Universal Robots PolyScope program: cov st move test.urp

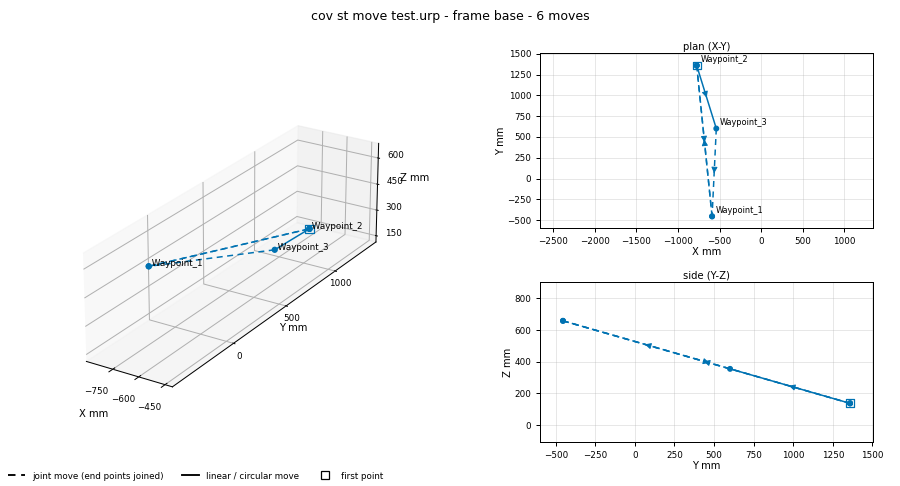
[picture p0: tool path of cov st move test.urp in frame base, 6 of 6 moves have a stored position in this frame; points joined in program order, loops and branches not executed]
Program cov st move test (installation=default directory=/programs createdIn=5.21.3 lastSavedIn=5.21.3 robotSerialNumber=20246801938)
Calibrated DH parameters: a=[-0.000071, -0.790281, -0.600694, 0.000061, -0.000039, 0]; d=[0.236272, 604.465945, 132.116513, -736.382239, 0.159268, 0.154005]; alpha=[1.570254, -0.000567, 0.000559, 1.571709, -1.56999, 0]; deltaTheta=[0, -0.409357, 7.293326, -0.600784, -0.000001, -0.000001]
InitVariablesNode
Robot Program (runOnlyOnce=false)
  Set NoAction tcp=pretend_w_top
  MoveL speed 250 mm/s, acceleration 1200 mm/s^2 (useActiveTCP=true optimoveEnabled=false optiMoveSpeed=0.3 optiMoveAcceleration=0.09) feature=Base
    Waypoint Waypoint_2: TCP in base x=-774.345 y=1358.868 z=137.57 mm, rx=1.008 ry=-1.4785 rz=-1.7543 rad; joints [-80.262, -40.663, 86.18, -52.649, 40.551, -3.676] deg; TCP offset x=-1.032 y=-18.062 z=285.234 mm, rx=0 ry=0 rz=0 rad
  If 1≟2
    MoveJ speed 60 deg/s, acceleration 80 deg/s^2 (useActiveTCP=true optimoveEnabled=false optiMoveSpeed=0.3 optiMoveAcceleration=0.09) feature=Base
      Waypoint Waypoint_1: TCP in base x=-589.354 y=-454.462 z=658.693 mm, rx=1.8664 ry=-1.8664 rz=-0.5984 rad; joints [32.16, -93.601, 92.579, 59.83, 108.044, 27.179] deg
      Waypoint Waypoint_2: TCP in base x=-774.345 y=1358.868 z=137.57 mm, rx=1.008 ry=-1.4785 rz=-1.7543 rad; joints [-80.262, -40.663, 86.18, -52.649, 40.551, -3.676] deg
  MoveL speed 250 mm/s, acceleration 1200 mm/s^2 (useActiveTCP=true optimoveEnabled=false optiMoveSpeed=0.3 optiMoveAcceleration=0.09) feature=Base
    Waypoint Waypoint_2: TCP in base x=-774.345 y=1358.868 z=137.57 mm, rx=1.008 ry=-1.4785 rz=-1.7543 rad; joints [-80.262, -40.663, 86.18, -52.649, 40.551, -3.676] deg
    Waypoint Waypoint_3: TCP in base x=-538.642 y=601.151 z=355.326 mm, rx=1.4044 ry=-1.6924 rz=-1.3263 rad; joints [-95.068, -88.736, 129.838, 12.913, 25.515, -61.155] deg
    SuppressedNode
      Waypoint Waypoint_1: TCP in base x=-589.354 y=-454.462 z=658.693 mm, rx=1.8664 ry=-1.8664 rz=-0.5984 rad; joints [32.16, -93.601, 92.579, 59.83, 108.044, 27.179] deg
  MoveJ speed 60 deg/s, acceleration 80 deg/s^2 (useActiveTCP=true optimoveEnabled=false optiMoveSpeed=0.3 optiMoveAcceleration=0.09) feature=Base
    Waypoint Waypoint_1: TCP in base x=-589.354 y=-454.462 z=658.693 mm, rx=1.8664 ry=-1.8664 rz=-0.5984 rad; joints [32.16, -93.601, 92.579, 59.83, 108.044, 27.179] deg
